PROGRAM PRG_LVCP2
VAR
END_VAR

	PRG_LVCP2_PowerMeasurement();

	PRG_LVCP2_CompensationCalculate();

	PRG_LVCP2_MainDisconnector();
	
	PRG_LVCP2_Colors();
	
	PRG_LVCP2_Group1();
	
	PRG_LVCP2_Group2();
	
	PRG_LVCP2_Group3();	
	
	PRG_LVCP2_Group4();	

	PRG_LVCP2_Group5();	

	PRG_LVCP2_Group6();	

	PRG_LVCP2_Group7();	

	PRG_LVCP2_Group8();	

	PRG_LVCP2_Group9();	

	PRG_LVCP2_Group10();

END_PROGRAM

(* stored: Version 1.1.0.1, ProductVersion 3.1.4024.14
   POU PRG_LVCP2: Id {8304e365-3362-440a-bc95-a318c3aca3b1}, SpecialFunc None *)
